
FUNCTION CB_dint_to_sint : INT

TITLE = ' Convert a double integer into an Int '
VERSION : '1.0'
AUTHOR  : CB
NAME    : DinToSin
FAMILY  : TNI

VAR_INPUT
    IN : DINT;
END_VAR

VAR_TEMP

END_VAR

BEGIN

CB_dint_to_sint := DINT_TO_INT(IN);

END_FUNCTION
